Yaskawa INFORM job: XYTRACE.JBI

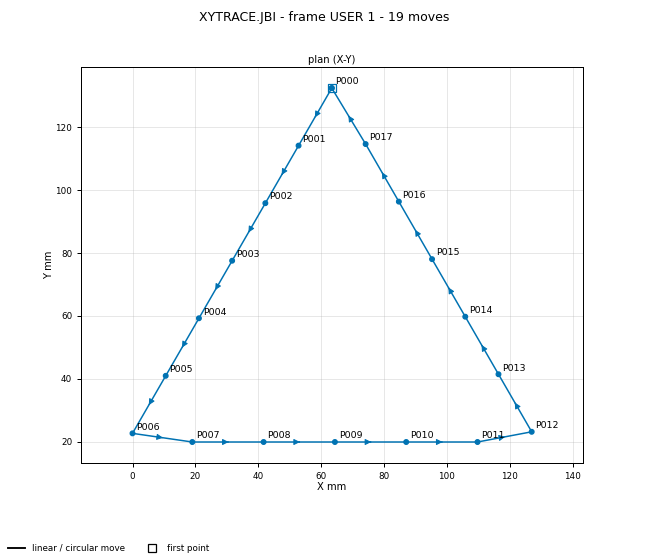
[picture p0: tool path of XYTRACE.JBI in frame USER 1, 19 of 19 moves have a stored position in this frame; points joined in program order, loops and branches not executed]
/JOB
//NAME XYTRACE
//POS
///NPOS 0,0,0,19,0,0
///USER 1
///TOOL 0
///POSTYPE USER
///RECTAN
///RCONF 0,0,0,0,0,0,0,0
P000=63.397,132.497,30.000,180.0000,0.0000,0.0000
P001=52.831,114.190,30.000,180.0000,0.0000,0.0000
P002=42.264,95.883,30.000,180.0000,0.0000,0.0000
P003=31.698,77.576,30.000,180.0000,0.0000,0.0000
P004=21.132,59.269,30.000,180.0000,0.0000,0.0000
P005=10.566,40.962,30.000,180.0000,0.0000,0.0000
P006=0.000,22.655,30.000,180.0000,0.0000,0.0000
P007=19.024,19.903,30.000,180.0000,0.0000,0.0000
P008=41.708,19.903,30.000,180.0000,0.0000,0.0000
P009=64.392,19.903,30.000,180.0000,0.0000,0.0000
P010=87.075,19.903,30.000,180.0000,0.0000,0.0000
P011=109.759,19.903,30.000,180.0000,0.0000,0.0000
P012=127.000,23.152,30.000,180.0000,0.0000,0.0000
P013=116.434,41.459,30.000,180.0000,0.0000,0.0000
P014=105.868,59.766,30.000,180.0000,0.0000,0.0000
P015=95.302,78.073,30.000,180.0000,0.0000,0.0000
P016=84.736,96.380,30.000,180.0000,0.0000,0.0000
P017=74.169,114.688,30.000,180.0000,0.0000,0.0000
P018=63.397,132.497,30.000,180.0000,0.0000,0.0000
//INST
///DATE 2026/04/08 12:00
///ATTR SC,RW
///GROUP1 RB1
NOP
MOVJ P000 VJ=5.00
MOVL P001 V=60.0
MOVL P002 V=60.0
MOVL P003 V=60.0
MOVL P004 V=60.0
MOVL P005 V=60.0
MOVL P006 V=60.0
MOVL P007 V=60.0
MOVL P008 V=60.0
MOVL P009 V=60.0
MOVL P010 V=60.0
MOVL P011 V=60.0
MOVL P012 V=60.0
MOVL P013 V=60.0
MOVL P014 V=60.0
MOVL P015 V=60.0
MOVL P016 V=60.0
MOVL P017 V=60.0
MOVL P018 V=60.0
END
